# EPICS substitutions: scopeApp/Db/ds6.substitutions
file mbbo3.db
{
pattern	{           DESC,        ITEM, N,  ZRST,    ONST,  TWST,    USER}
	{    "Trig Mode",   TRIG:MODE, 0,  Edge,   Pulse, Slope,  TRMODE}
	{   "Trig Sweep",  TRIG:SWEEP, 0,  Auto,  Normal,Single,   TRSWE}
	{   "Trig Slope",  TRIG:SLOPE, 0,  Rise,    Fall, RFall,   TRSLO}
	{"Time Ref Mode",TIME:HR:MODE, 0, Center,TrigPos,  User, TMHMODE}
	{    "Time Mode",   TIME:MODE, 0,   Main,     XY,  Roll,  TMMODE}
}
file mbbo4.db
{
pattern	{          DESC,     ITEM, N,   ZRST,    ONST, TWST,   THST,   USER}
	{  "Time Div U",TIM:DIV:U, 0,     ns,      us,   ms,    sec,TIMDIVU}
	{  "Trig Coupl", TRIG:CPL, 0,     AC,      DC,  LFR,    HRF,  TRCPL}
	{ "AcquireType", ACQ:TYPE, 0, Normal,Averages, Peak, HResol,  ACQTP}
}
file bo.db
{
pattern	{          DESC,      ITEM, N,    ZNAM,   ONAM,  USER}
	{  "Auto Scale",AUTO:SCALE, 0, AutoScl,AutoScl, AUTOS}
	{   "WF Format",    WF:FMT, 0,    Byte,   Word, WFFMT}
	{  "Time XY 12", TIME:XY12, 0,     Off,     On, TMXY1}
	{  "Time XY 34", TIME:XY34, 0,     Off,     On, TMXY2}
}
file lo.db
{
pattern	{             DESC,      ITEM, LOPR, HOPR,    USER}
	{  "TBase Scale V",TIME:DIV:V,    0,    0, TIMDIVV}
	{   "SRE register",       SRE,    0,    0,     SRE}
	{ "SampleAverages",  ACQ:AVRG,    1, 9999,   ACQAV}
}
file ao.db
{
pattern {             DESC,     ITEM, N,  DRVL, DRVH,  EGU,    USER}
	{    "TBase Scale", TIME:DIV, 0,     0,    0,s/div,  TIMDIV}
	{   "TBase Offset",TIME:OFST, 0,     0,    0,s/div,  TMOFST}
	{"TBase Dly Scale",TIME:DSCL, 0,     0,    0,s/div,TMDLYSCL}
}
file si.db
{
pattern	{         DESC,      ITEM, N,  USER}
	{ "Sampl Rate", SMPL:RATE, 0, SRATE}
	{ "Trig State",TRIG:STATE, 0, TRSTA}
}
file scopeTrace.db
{
pattern { N, NELM}
        { 0, 1400}
        { 1, 1400}
        { 2, 1400}
        { 3, 1400}
}
file ds6Ctrl.db{
  {N=0}
}
